// TwinCAT 3 PLC project SmartHome_OfUncleSasha
// ProgramVersion: 3.1.4026.20
// CompilerDefines: VISU_USEPROPERTYINFO
// libraries:
//   [Smart Home Device Library], * (Oleksandr Tiutyk)
//   [Smart Home Library], * (Oleksandr Tiutyk)
//   Tc2_Standard, * (Beckhoff Automation GmbH)
//   Tc2_System, * (Beckhoff Automation GmbH)
//   VisuDialogs, * (System)
// project tree:
//   / GlobalTextList.TcGTLO, MAIN.TcPOU, PlcTask.TcTTO, SmartHomeOfUncleSasha.TcPOU, Visualization Manager.TcVMO (not stored), Visualization.TcVIS
// (motion and I/O tree: see PLC project smarthome_referencelibrary)
// real-time tasks:
//   TASK PlcTask: cycle T#10ms, priority 20, ADS port 350
//   TASK PlcTask1: cycle T#10ms, priority 21, ADS port 351

CONFIGURATION SmartHome_OfUncleSasha
    RESOURCE PLC ON TwinCAT3
        TASK PlcTask(INTERVAL := T#10ms, PRIORITY := 20);
        PROGRAM MAIN WITH PlcTask : MAIN;
    END_RESOURCE
END_CONFIGURATION

// ---- MAIN.TcPOU
PROGRAM MAIN
VAR
	SmartHome : SmartHomeOfUncleSasha;
	
	Home : REFERENCE TO SHLib.SmartHome<5>; 
END_VAR

IF NOT __ISVALIDREF(Home) THEN	
	Home REF= SmartHome; 
END_IF

Home.Execute();

END_PROGRAM

// ---- SmartHomeOfUncleSasha.TcPOU
FUNCTION_BLOCK SmartHomeOfUncleSasha EXTENDS SmartHome<5>
VAR
	CarbonDioxideSensor_Room_1 : SHDevLib.CarbonDioxideSensor('Room 1');
	Ventilation_Room_1 : SHDevLib.Ventilation('Room 1');

	CarbonDioxideSensor_Kitchen : SHDevLib.CarbonDioxideSensor('Kitchen');
	Ventilation_Kitchen : SHDevLib.Ventilation('Kitchen');
	
	ClimatSystem_Room_1 : SHDevLib.ClimatSystem('Room 1');
END_VAR

METHOD PROTECTED GetDeviceArray : ARRAY [0.._DeviceCount - 1] OF IDevice
GetDeviceArray[0] := CarbonDioxideSensor_Room_1;
GetDeviceArray[1] := Ventilation_Room_1;

GetDeviceArray[2] := CarbonDioxideSensor_Kitchen;
GetDeviceArray[3] := Ventilation_Kitchen;
	
GetDeviceArray[4] := ClimatSystem_Room_1;
END_METHOD

METHOD PROTECTED OnTick
IF CarbonDioxideSensor_Room_1.CarbonDioxideLevel > 1100 THEN
	Ventilation_Room_1.SetSpeed(3);
ELSIF CarbonDioxideSensor_Room_1.CarbonDioxideLevel > 900 THEN
	Ventilation_Room_1.SetSpeed(2);
ELSIF CarbonDioxideSensor_Room_1.CarbonDioxideLevel > 700 THEN
	Ventilation_Room_1.SetSpeed(1);
ELSE
	Ventilation_Room_1.SetSpeed(0);
END_IF

IF CarbonDioxideSensor_Kitchen.CarbonDioxideLevel > 1200 THEN
	Ventilation_Kitchen.SetSpeed(3);
ELSIF CarbonDioxideSensor_Kitchen.CarbonDioxideLevel > 1000 THEN
	Ventilation_Kitchen.SetSpeed(2);
ELSIF CarbonDioxideSensor_Kitchen.CarbonDioxideLevel > 800 THEN
	Ventilation_Kitchen.SetSpeed(1);
ELSE
	Ventilation_Kitchen.SetSpeed(0);
END_IF

SUPER^.OnTick();
END_METHOD

END_FUNCTION_BLOCK

// ---- GlobalTextList.TcGTLO
TEXTLIST GlobalTextList
  463 = '> 1100 => 3 , > 900 => 2, > 700 => 1, ELSE 0'
  11 = '> 1200 => 3 , > 1000 => 2, > 800 => 1, ELSE 0'
  453 = 'Alarm'
  347 = 'Alarm system (door)'
  714 = 'Alarm system (door):'
  336 = 'Carbon dioxide sensor error'
  982 = 'Carbon dioxide value'
  811 = 'Carbon dioxide value %4f'
  290 = 'Carbon dioxide value: %4f'
  117 = 'Carbon dioxide value: %d'
  660 = 'Climat system error'
  335 = 'Cooling ON'
  581 = 'Cooling ON (>= 30)'
  954 = 'Cooling ON (t >= 30)'
  746 = 'Error'
  544 = 'Heating ON'
  205 = 'Heating ON (<= 20)'
  156 = 'Heating ON (t <= 20)'
  992 = 'Kitchen'
  648 = 'Room 1'
  208 = 'Temperature value: %2f'
  495 = 'Temperature value: %d'
  196 = 'Ventilation error'
  341 = 'Ventilation fan speed: %2f'
  614 = 'Ventilation fan speed: %d'
END_TEXTLIST

// ---- Visualization.TcVIS
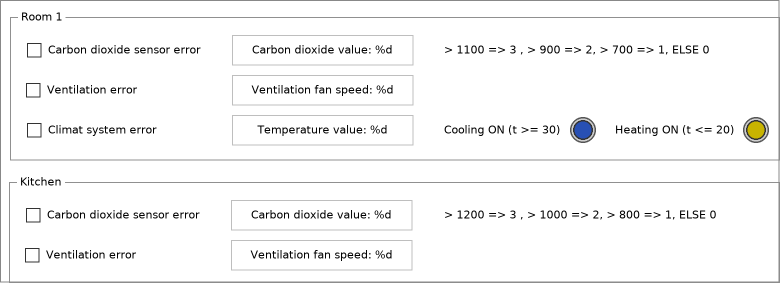
VISUALIZATION Visualization  // 780x283
    GroupBox (10,9 770x151), "Room 1"
        Checkbox (15,26 192x30), "Carbon dioxide sensor error", variable: MAIN.SmartHome.CarbonDioxideSensor_Room_1.ErrorSimulation
        Checkbox (14,66 193x30), "Ventilation error", variable: MAIN.SmartHome.Ventilation_Room_1.ErrorSimulation
        Checkbox (15,106 191x30), "Climat system error", variable: MAIN.SmartHome.ClimatSystem_Room_1.ErrorSimulation
        Textfield (222,26 181x30), "Carbon dioxide value: %d", text variable: MAIN.SmartHome.CarbonDioxideSensor_Room_1._CarbonDioxideLevel
            OnMouseClick: write the text variable via Default
        Textfield (222,66 181x30), "Ventilation fan speed: %d", text variable: MAIN.SmartHome.Ventilation_Room_1._Speed
        Textfield (222,106 181x30), "Temperature value: %d", text variable: MAIN.SmartHome.ClimatSystem_Room_1._Temperature
            OnMouseClick: write the text variable via Default
        Label (431,106 120x30), "Cooling ON (t >= 30)"
        Lamp1 (553,106 40x30), variable: MAIN.SmartHome.ClimatSystem_Room_1._IsCoolingOn, style: Lamp-Lamp1-Blue
        Label (602,106 123x30), "Heating ON (t <= 20)"
        Lamp1 (726,106 40x30), variable: MAIN.SmartHome.ClimatSystem_Room_1._IsHeatingOn, style: Lamp-Lamp1-Yellow
        Label (431,26 328x30), "> 1100 => 3 , > 900 => 2, > 700 => 1, ELSE 0"
    GroupBox (9,174 771x109), "Kitchen"
        Checkbox (15,26 192x30), "Carbon dioxide sensor error", variable: MAIN.SmartHome.CarbonDioxideSensor_Kitchen.ErrorSimulation
        Checkbox (14,66 193x30), "Ventilation error", variable: MAIN.SmartHome.Ventilation_Kitchen.ErrorSimulation
        Textfield (222,26 181x30), "Carbon dioxide value: %d", text variable: MAIN.SmartHome.CarbonDioxideSensor_Kitchen._CarbonDioxideLevel
            OnMouseClick: write the text variable via Default
        Textfield (222,66 181x30), "Ventilation fan speed: %d", text variable: MAIN.SmartHome.Ventilation_Kitchen._Speed
        Label (432,26 328x30), "> 1200 => 3 , > 1000 => 2, > 800 => 1, ELSE 0"
END_VISUALIZATION
